FUNCTION_BLOCK MECH2_PRXY (* Proxy for a Remote Bidirectional Mechanism *)
  (* Standard: 61499-1 *)
  (* Version 0.0, 2004-09-26, JHC, Rockwell Automation *)
  (* Compiler header: package fb.rt.mva; import fb.rt.net.*; *)
  (* Compiler Java Sun JDK 1.4.2 *)
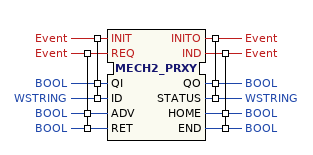
  EVENT_INPUT
    INIT WITH QI, ID; (* Initialize Client/Server Connection *)
    REQ WITH ADV, RET; (* Send Actuator Data *)
  END_EVENT
  EVENT_OUTPUT
    INITO WITH QO, STATUS; (* INIT Acknowledgment *)
    IND WITH HOME, END; (* Sensor Change Indication *)
  END_EVENT
  VAR_INPUT
    QI : BOOL; (* Event Input Qualifier *)
    ID : WSTRING; (* Connection Identifier *)
    ADV : BOOL; (* ADVANCE *)
    RET : BOOL; (* RETRACT *)
  END_VAR
  VAR_OUTPUT
    QO : BOOL; (* Event Output Qualifier *)
    STATUS : WSTRING; (* Service Status *)
    HOME : BOOL; (* HOME Position Sensor *)
    END : BOOL; (* END Position Sensor *)
  END_VAR
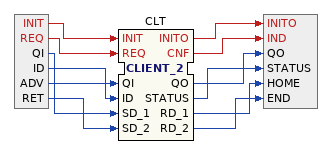
  FBS
    CLT : CLIENT_2;
  END_FBS
  EVENT_CONNECTIONS
    INIT TO CLT.INIT;
    CLT.INITO TO INITO;
    CLT.CNF TO IND;
    REQ TO CLT.REQ;
  END_CONNECTIONS
  DATA_CONNECTIONS
    QI TO CLT.QI;
    CLT.QO TO QO;
    ID TO CLT.ID;
    CLT.STATUS TO STATUS;
    ADV TO CLT.SD_1;
    CLT.RD_1 TO HOME;
    RET TO CLT.SD_2;
    CLT.RD_2 TO END;
  END_CONNECTIONS
END_FUNCTION_BLOCK
